PROGRAM MAIN
VAR
	START  : BOOL;
	STOP   : BOOL;
	EMERG  : BOOL := TRUE;
	ACK    : BOOL;
	MASTER : MASTER;
END_VAR

MASTER(START := START, STOP := STOP, EMERG := EMERG, ACK := ACK);

END_PROGRAM

(* stored: Version 1.1.0.1, ProductVersion 3.1.4024.12
   POU MAIN: Id {ee4bee94-b289-42a5-ba7b-d84e1810ac9a}, SpecialFunc None *)
